KUKA KRL program: chk_w4_wechs_ok.src

&ACCESS RVO9
&REL 1
&COMMENT Check C3
DEF chk_w4_wechs_ok( )
;Diag_Appl(#on,5)

; VERIFICAÇÃO DE FERRAMENTA: C3

$TIMER[10] = 0
$TIMER_STOP[10] = FALSE

wait for (($in[161]) and (($in[169]) or (NOT ($in[169]) and $in[3320])) and ($in [177]) and (NOT $in [185]) and ( $in[219]))

$TIMER_STOP[10] = TRUE
$TIMER[10] = 0

;//---- End -------
;Diag_Appl(#Off,5)
END
